{attribute 'TcGenerated'}
{attribute 'no-analysis'}
{attribute 'linkalways'}
// This function has been automatically generated from the project information.
VAR_GLOBAL CONSTANT
	{attribute 'const_non_replaced'}
	stLibVersion_TcUnit_Zeugwerk : ST_LibVersion := (iMajor := 1, iMinor := 3, iBuild := 2, iRevision := 0, nFlags := 0, sVersion := '1.3.2');
END_VAR

(* stored: Version 1.1.0.1
   GVL Global_Version: Id {899e68fc-21fd-4d89-beb5-fc369f4dda74} *)
